RoboDK station: dld.rdk

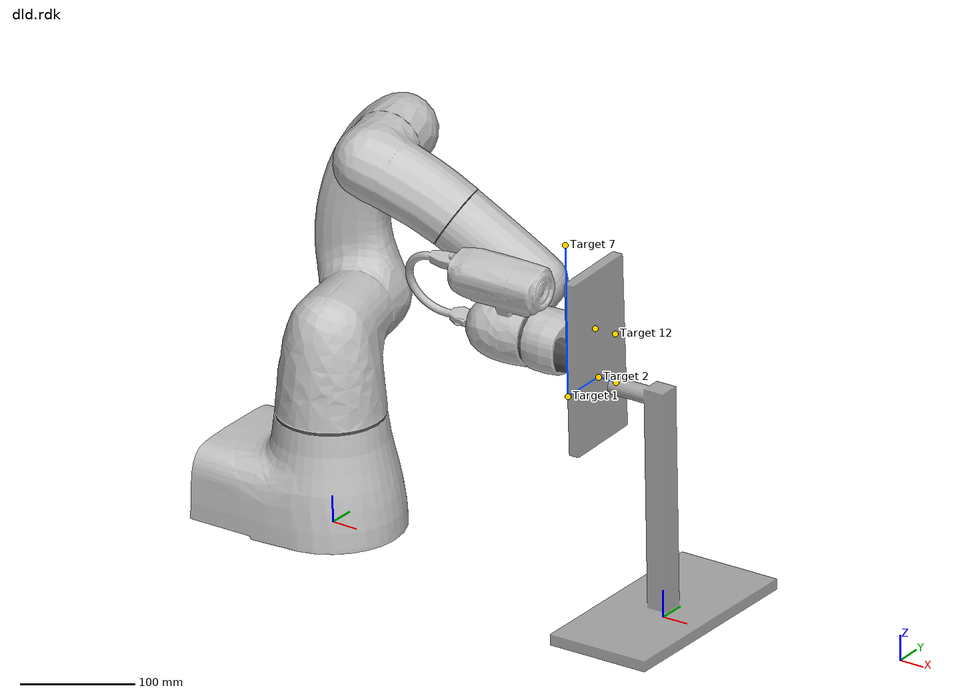
[picture v0: the station drawn from its stored meshes, robots at their saved joint values, targets as dots, program paths as lines]
Station dld (saved by RoboDK 5.6.0). Poses are relative to the parent item; angles as X-Y-Z fixed-axis rotations.
Station parameters (name, value as stored): LIN64
  - frame Denso Cobotta Base at (0, 0, 0) mm, rotated rx 0 ry -1.03 rz 0 deg
    - robot Denso Cobotta: 6 axes, payload 4 kg, reach 342.5 mm, repeatability 0.05 mm, weight 29 kg
        modified DH rows (alpha deg, a mm, theta deg, d mm): 0, 0, 0, 180; -90, 0, -90, 20; 0, 165, -90, 0; -90, 12, 0, 177.5; 90, 0, 0, -64.5; -90, 0, 0, 102
        joint limits [-150, -60, -18, -170, -95, -170] to [150, 100, 140, 170, 135, 170]; home [0, 0, 90, 0, 0, 0]; saved at [12.413, 11.2, 112.203, 19.7, -35.315, -15.524]
      - tool smartphone2, TCP at (0, 0, 4.49) mm, size 165 x 76 x 10 mm, geometry from smartphone2.stl
    - frame Frame 2 at (350, 0, 0) mm
      - object suporte at (0, 0, 0) mm, size 100 x 200 x 220 mm, geometry from suporte.stl
      - target Target 7 (Cartesian target) at (-66.01, -44.5, 357) mm, rotated rx -180 ry 90 rz -180 deg; joints [0, 0, 90, 0, -0.004, 0] of Denso Cobotta
      - target Target 1 (Cartesian target) at (-66.01, -44.5, 212.12) mm, rotated rx -180 ry 90 rz -180 deg; joints [0, 17.924, 120.522, 0, -48.445, 0] of Denso Cobotta
      - target Target 2 (Cartesian target) at (-66.01, 1.74, 212.12) mm, rotated rx -178.86 ry 90 rz -178.86 deg; joints [13.765, 16.666, 115.13, 20.182, -43.605, -14.904] of Denso Cobotta
      - target Target 3 (Cartesian target) at (-47.3, 1.74, 212.12) mm, rotated rx -177.74 ry 90 rz -177.74 deg; joints [12.552, 21.937, 107.99, 19.132, -41.536, -14.557] of Denso Cobotta
      - target Target 4 (Cartesian target) at (-66.01, 1.74, 212.12) mm, rotated rx -178.22 ry 90 rz -178.22 deg; joints [13.765, 16.666, 115.13, 20.182, -43.605, -14.904] of Denso Cobotta
      - target Target 5 (Cartesian target) at (-66.01, -44.5, 212.12) mm, rotated rx -180 ry 90 rz -180 deg; joints [0, 17.924, 120.522, 0, -48.445, 0] of Denso Cobotta
      - target Target 6 (Cartesian target) at (-66.01, -44.5, 357) mm, rotated rx -180 ry 90 rz -180 deg; joints [0, 0, 90, 0, -0.004, 0] of Denso Cobotta
      - target Target 8 (Cartesian target) at (-66.01, -44.5, 356.99) mm, rotated rx -180 ry 90 rz -180 deg; joints [0, 0, 89.999, 0.003, 0.006, -0.003] of Denso Cobotta
      - target Target 9 (Cartesian target) at (-66.01, -44.5, 212.12) mm, rotated rx 0 ry 90 rz 0 deg; joints [0, 17.924, 120.522, 0, -48.446, 0] of Denso Cobotta
      - target Target 10 (Cartesian target) at (-66.01, 1.74, 212.12) mm, rotated rx -180 ry 90 rz -180 deg; joints [13.765, 16.666, 115.13, 20.182, -43.605, -14.904] of Denso Cobotta
      - target Target 11 (Cartesian target) at (-47.3, 1.74, 212.12) mm, rotated rx 0 ry 90 rz 0 deg; joints [12.552, 21.937, 107.99, 19.132, -41.536, -14.557] of Denso Cobotta
      - target Target 12 (Cartesian target) at (-47.3, 1.74, 258.41) mm, rotated rx -0.07 ry 90 rz -0.07 deg; joints [11.298, 12.135, 99.53, 28.42, -24.307, -26.252] of Denso Cobotta
      - target Target 13 (Cartesian target) at (-68.61, 1.74, 258.41) mm, rotated rx 0.06 ry 90 rz 0.06 deg; joints [12.375, 5.067, 107.135, 30.142, -25.264, -27.705] of Denso Cobotta
      - target Target 14 (Cartesian target) at (-66.01, -44.5, 357.01) mm, rotated rx 0 ry 90 rz 0 deg; joints [0, 0.001, 89.991, 0.024, 0.004, -0.024] of Denso Cobotta
  - program Touch (9 instructions, listed below)
  - Python program Prog2 (listed below)
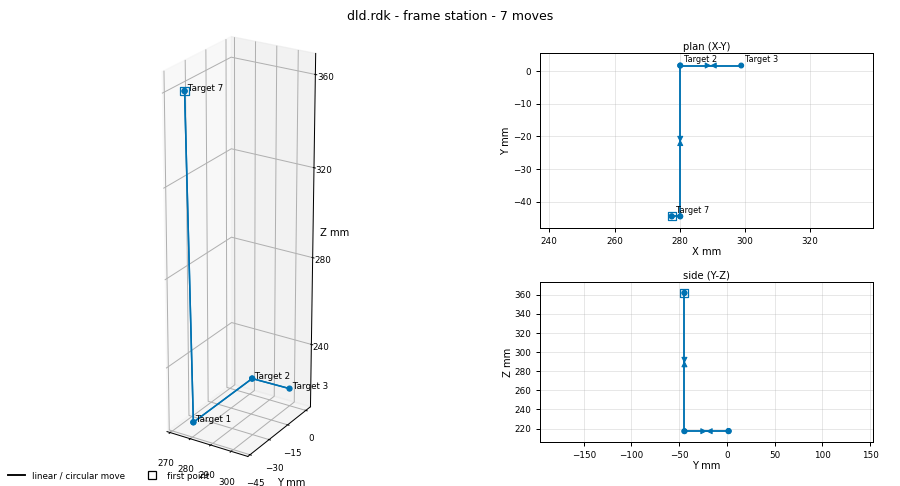
[picture p0: tool path of dld.rdk in frame station, 7 of 7 moves have a stored position in this frame; points joined in program order, loops and branches not executed]

--- program Touch (robot Denso Cobotta) ---
  Set Ref.: Frame 2
  MoveL (Target 7)
  Set Tool: smartphone2
  MoveL (Target 1)
  MoveL (Target 2)
  MoveL (Target 3)
  MoveL (Target 4)
  MoveL (Target 5)
  MoveL (Target 6)

--- Python program Prog2 ---
# Type help("robodk.robolink") or help("robodk.robomath") for more information
# Press F5 to run the script
# Documentation: https://robodk.com/doc/en/RoboDK-API.html
# Reference:     https://robodk.com/doc/en/PythonAPI/robodk.html
# Note: It is not required to keep a copy of this file, your Python script is saved with your RDK project

# You can also use the new version of the API:
from robodk import robolink    # RoboDK API
from robodk import robomath    # Robot toolbox
RDK = robolink.Robolink()

# Forward and backwards compatible use of the RoboDK API:
# Remove these 2 lines to follow python programming guidelines
from robodk import *      # RoboDK API
from robolink import *    # Robot toolbox
# Link to RoboDK
# RDK = Robolink()

# Notify user:
print('To edit this program:\nright click on the Python program, then, select "Edit Python script"')

# Program example:
item = RDK.Item('base')
if item.Valid():
    print('Item selected: ' + item.Name())
    print('Item posistion: ' + repr(item.Pose()))

print('Items in the station:')
itemlist = RDK.ItemList()
print(itemlist)

# Provoking an exception will display the console output if you run this script from RoboDK
raise Exception('Program not edited.')
